// TIA Portal V20 export
// export: Created 2026-10-06T14:29:35.2795735Z, ExportSetting WithDefaults, DisplayName Totally Integrated Automation Portal, DisplayVersion V20, DisplayName TIA Portal Openness, DisplayVersion V20, DisplayName TIA Portal Version Control Interface, DisplayVersion V20, DisplayName SINAMICS Startdrive Advanced, DisplayVersion V20, DisplayName SINAMICS Startdrive G130, G150, S120, S150, SINAMICS MV, G220, S200, S210, DisplayVersion V20, DisplayName SINAMICS Startdrive G110M, G120, G120C, G120D, G120P, G115D, DisplayVersion V20, DisplayName STEP 7 Professional, DisplayVersion V20, DisplayName STEP 7 Safety, DisplayVersion V20, DisplayName WinCC Basic/Comfort/Advanced, DisplayVersion V20, DisplayName WinCC Unified, DisplayVersion V20
FUNCTION_BLOCK "MotorSequenceLAD"   // FB1, SCL
{ S7_Optimized_Access := 'TRUE' }
VERSION : 2.0
// stored: AutoNumber true, IsIECCheckEnabled false, IsRetainMemResEnabled false, MemoryReserve 100, SetENOAutomatically false, UDAEnableTagReadback false
   VAR_INPUT
      Start : Bool;
      Stop : Bool;
      StartInterval : Time;
      StopInterval : Time;
   END_VAR
   VAR_OUTPUT
      Motor1 : Bool;
      Motor2 : Bool;
      Motor3 : Bool;
      Stopping : Bool;
   END_VAR
   VAR
      Active1 : Bool;
      Active2 : Bool;
      Active3 : Bool;
      PreviousStart : Bool;
      StartPulse : Bool;
      StopEvent : Bool;
      Had3 : Bool;
      Had2 : Bool;
      Start2Done : Bool;
      Start3Done : Bool;
      Stop2Done : Bool;
      Stop1Done : Bool;
      Start2 { S7_SetPoint := 'True'} : TON_TIME;
      Start3 { S7_SetPoint := 'True'} : TON_TIME;
      Stop2 { S7_SetPoint := 'True'} : TON_TIME;
      Stop1 { S7_SetPoint := 'True'} : TON_TIME;
   END_VAR
BEGIN

   #Start2(IN := FALSE,
           PT := #StartInterval);
   #Start3(IN := FALSE,
           PT := #StartInterval);
   #Stop2(IN := FALSE,
          PT := #StopInterval);
   #Stop1(IN := FALSE,
          PT := #StopInterval);
END_FUNCTION_BLOCK
